//{attribute 'qualified_only'}
VAR_GLOBAL
	
	
END_VAR

(* stored: Version 1.1.0.1, ProductVersion 3.1.4024.12
   GVL GVL_AXES: Id {91bd79a2-50f8-44b0-96e4-bd73e085d622} *)
